// TwinCAT 3 PLC project HalfBROT
// Title: HalfBROT
// Company: BROT
// ProjectVersion: 0.4.4
// ProgramVersion: 3.1.4024.66
// CompilerDefines: VISU_USEPROPERTYINFO
// libraries:
//   AstroBROT, * (BROT)
//   BROTLib, * (BROT)
//   Tc2_MC2, * (Beckhoff Automation GmbH)
//   Tc2_MC2_Drive, * (Beckhoff Automation GmbH)
//   Tc2_Standard, * (Beckhoff Automation GmbH)
//   Tc2_System, * (Beckhoff Automation GmbH)
//   Tc2_Utilities, * (Beckhoff Automation GmbH)
//   Tc3_Module, * (Beckhoff Automation GmbH)
//   VisuDialogs, * (System)
//   VisuSymbols, * (System)
//   VisuSymbols,3.5.10.0,System
// project tree:
//   / GlobalTextList.TcGTLO, VisualizationManager.TcVMO (not stored)
//   POUs/ FB_AxisControl.TcPOU, FB_AzimuthControl.TcPOU, FB_CoverControl.TcPOU, FB_DerotatorControl.TcPOU, FB_ElevationControl.TcPOU, FB_FocusControl.TcPOU, FB_HydraulicsControl.TcPOU, FB_PendantControl.TcPOU, FB_TelescopeAuxiliary.TcPOU
//   VISUs/ Azimuth.TcVIS, Cover.TcVIS, Derotator.TcVIS, Elevation.TcVIS, Focus.TcVIS, Hydraulics.TcVIS
//   GVLs/ Global_Version.TcGVL

// ---- GVLs/Global_Version.TcGVL
{attribute 'qualified_only'}
VAR_GLOBAL CONSTANT
	// Mirrors Beckhoff's own Global_Version.stLibVersion_* pattern (see ST_LibVersion),
	// which only covers Tc2_*/Tc3_* library references, not custom ones -- until now: this
	// GVL uses Beckhoff's own naming exactly, so it merges into a consumer's Global_Version.
	// Kept in sync with <ProjectVersion> in HalfBROT.plcproj at release time.
	stLibVersion_HalfBROT : ST_LibVersion := (
		iMajor := 0,
		iMinor := 4,
		iBuild := 4,
		iRevision := 0,
		nFlags := 1,
		sVersion := '0.4.4'
	);
END_VAR

// ---- POUs/FB_AxisControl.TcPOU
FUNCTION_BLOCK ABSTRACT FB_AxisControl EXTENDS FB_BaseAxis IMPLEMENTS I_Axis
VAR_INPUT
	bMoveAxis				: BOOL;		// Move azimuth to given position
	bTracking				: BOOL;		// enable tracking
	bStopAxis				: BOOL;		// stop the Axis
	fMinPosition			: REAL := 0;
	fMaxPosition			: REAL := 450.0;
	fCalibPosition			: LREAL := 45.0; // // current position of the calibration cam
END_VAR
VAR_OUTPUT
END_VAR
VAR
	fSlewTime				: LREAL;	// time to reach target position

	InDigitalInputs	  AT%I*	: WORD;		// digitale inputs der Endlagen
	InDiagnostic	  AT%I*	: UDINT;	// diagnostic number
	InTorque	 	  AT%I*	: INT;		// derotator torque feedback
	IbSTO		  	  AT%I*	: BOOL;		// STO

	fbAxisCalibration		: MC_SetPosition;

	axisEvent			: FB_EventLog;
	diagnosticEvent		: FB_EventLog;
	
	bDiagnosticError		: BOOL;
	
	fbReadParameter		: MC_ReadParameter;
	bGetLastPosition		: BOOL := TRUE;
	
	calibrationEvent		: FB_Eventlog;
	fTorque			: REAL;	// percentage of the derotator torque
	torqueWarning			: FB_EventLog;	
END_VAR
VAR PERSISTENT
	fLastPosition			: LREAL := -1.0;
END_VAR

PROPERTY isTracking : BOOL
GET
isTracking := fbAxis.isTracking;
END_GET
END_PROPERTY

PROPERTY MoveAxis : BOOL
GET
MoveAxis := bMoveAxis;
END_GET
SET
bMoveAxis := MoveAxis;
END_SET
END_PROPERTY

PROPERTY MoveDone : BOOL
GET
MoveDone := fbAxis.MoveDone;
END_GET
END_PROPERTY

PROPERTY SlewTime : LREAL
GET
SlewTime := fSlewTime;
END_GET
END_PROPERTY

PROPERTY StopAxis : BOOL
GET
StopAxis := bStopAxis;
END_GET
SET
bStopAxis := StopAxis;
END_SET
END_PROPERTY

PROPERTY Tracking : BOOL
GET
Tracking := bTracking;
END_GET
SET
bTracking := Tracking;
END_SET
END_PROPERTY

END_FUNCTION_BLOCK

// ---- POUs/FB_AzimuthControl.TcPOU
FUNCTION_BLOCK FB_AzimuthControl EXTENDS FB_AxisControl
VAR_INPUT
	bBrakeOpen				: BOOL;		// azimuth break is open
END_VAR
VAR_OUTPUT
END_VAR
VAR
	tonReadyDelay		: TON;		// delay until commutator angle is measured
	homeDelay			: FB_TONTP;
	tonTorqueError		: TON := (PT := T#3S);
	tonRestTimer			: TON;
	bAtRest				: BOOL;
END_VAR

(* Azimuth Axis control section
Power must be on and brake must be open for the axis to operate
*)

// generate the ready signal after enabling the drive
tonReadyDelay(IN :=  fbAxis.Enable, PT := T#3000MS, Q=> bReady);

// limit the input position angle
fPosition := LIMIT(fMinPosition, fPosition, fMaxPosition);

// conduct the calibrated signal
bCalibrated := fbAxis.Calibrated;

IF bCalibrated OR bError THEN
	bHomeAxis := FALSE;
	bGetLastPosition := FALSE;
END_IF
	
IF bHomeAxis THEN
	fPosition := fCalibPosition;
END_IF

IF homeDelay.Q THEN
	fPosition := fCalibPosition;
	bMoveAxis := TRUE;
END_IF

// perform a recalibration on the last known position
fbAxisCalibration(
	Axis 		:= axisRef,
	Execute 	:= bGetLastPosition AND fLastPosition>=0.0 AND NOT bCalibrated,
	Position 	:= fLastPosition);

IF fbAxisCalibration.Done THEN
	bGetLastPosition := FALSE;
END_IF

IF bCalibrated THEN
	fLastPosition := fActualPosition;
END_IF

// enable the azimuth if not moved by the power chain. Sorry for the hack
tonRestTimer(IN := bBrakeOpen AND (ABS(axisRef.NcToPlc.ActVelo) < 0.01), PT := T#2S);
// if azimuth at rest or calibrated, allow enabling the azimuth (the brake must still be open, see Enable below)
IF tonRestTimer.Q or bCalibrated THEN
	bAtRest := TRUE;
ELSIF NOT bBrakeOpen THEN
	bAtRest := FALSE;
END_IF
	
// deactivate limit switches on homing
MC_SetAcceptBlockedDriveSignal(
	Axis 	:= axisRef, 
	Enable 	:= bHomeAxis);

fbAxis(	
	Enable 			:= bEnable AND bAtRest AND bBrakeOpen,
	Reset 			:= bReset,
	MoveAxis 		:= bMoveAxis,
	HomeAxis 		:= bHomeAxis,
	StopAxis 		:= bStopAxis,
	Tracking 		:= bTracking,
	Position 		:= fPosition, 
	Velocity 		:= fVelocity,
	Enable_Positive := inDigitalInputs.1 OR bHomeAxis,
	Enable_Negative := inDigitalInputs.0,
	Jog_Forward 	:= bMovePos,
	Jog_Backwards 	:= bMoveNeg,
	bCalibrationCam := NOT inDigitalInputs.1,
	ActualPosition 	=> fActualPosition,
	Error 			=> bError,
	ErrorID 		=> nErrorID,
	AxisRef 		:= axisRef);

IF bSoEReset THEN
	fLastPosition := -1.0;
	fbSoEReset(
		Axis 	:= axisRef,
		Execute := TRUE,
		Timeout := DEFAULT_ADS_TIMEOUT);
 	IF fbSoEReset.Busy THEN
		fbSoEReset(Axis := axisRef, Execute := FALSE);
	ELSE
		bSoEReset := FALSE;
		bReset := TRUE;
	END_IF
END_IF 

IF fbAxis.MoveDone THEN
	bMoveAxis := FALSE;
END_IF

IF fbAxis.HomeDone THEN
	bHomeAxis := FALSE;
END_IF
	
IF fbAxis.ResetDone THEN
	bReset := FALSE;
END_IF

IF fbAxis.StopDone THEN
	bStopAxis := FALSE;
END_IF
bDiagnosticError := FALSE;
IF inDiagnostic < 16#D012 AND inDiagnostic > 16#D014 THEN
	bDiagnosticError :=TRUE;
	nErrorID := inDiagnostic;
END_IF

fbReadParameter(	
	Axis 			:= axisRef, 
	Enable 			:= fbAxis.InMotion, 
	ParameterNumber := MC_AxisParameter.AxisRemainingTimeToGo, 
	ReadMode 		:= E_ReadMode.READMODE_CYCLIC);
IF fbReadParameter.Valid THEN
	fSlewTime := fbReadParameter.Value;
END_IF

fTorque := inTorque / 10.0;
tonTorqueError(IN := ABS(fTorque) > 50.0);

axisEvent(	
	Trigger 		:= bError, 
	Level 			:= ADSLOG_MSGTYPE_ERROR,
	FormatString 	:= 'Azimuth Axis Error: %s',
	OnMessage 		:= NCError_TO_STRING(nErrorID),
	Comm 			:= fbComm);
	
diagnosticEvent(	
	Trigger 		:= bDiagnosticError,
	Level 			:= ADSLOG_MSGTYPE_ERROR,
	FormatString 	:= 'Azimuth Axis Diagnostic Error: %s',
	OnMessage 		:= NCError_TO_STRING(inDiagnostic),
	Comm 			:= fbComm);
	
TorqueWarning(	
	Trigger 		:= tonTorqueError.Q, 
	Level 			:= ADSLOG_MSGTYPE_WARN,
	FormatString 	:= '%s',
	OnMessage 		:= 'Azimuth torque is high.',
	Comm 			:= fbComm);
	
CalibrationEvent(
	Trigger 		:= bCalibrated, 
	Level 			:= ADSLOG_MSGTYPE_HINT,
	FormatString 	:= '%s',
	OnMessage 		:= 'Azimuth axis is calibrated.',
	Comm 			:= fbComm);

PROPERTY InNegLimit : BOOL
GET
InNegLimit := NOT inDigitalInputs.0;
END_GET
END_PROPERTY

PROPERTY InPosLimit : BOOL
GET
InPosLimit := NOT inDigitalInputs.1;
END_GET
END_PROPERTY

END_FUNCTION_BLOCK

// ---- POUs/FB_CoverControl.TcPOU
FUNCTION_BLOCK FB_CoverControl IMPLEMENTS I_MirrorCovers
VAR_INPUT
	// output signals for opening/closing covers	
	OabOpenCover  AT%Q* : ARRAY[1..3] OF BOOL;	// open cover1-3 command
	OabCloseCover AT%Q* : ARRAY[1..3] OF BOOL;   // close cover1-3 command
	
	// telemetry interval
	fTelemetryInterval		: TIME := T#5S;	
END_VAR
VAR_OUTPUT
	bAllOpen			: BOOL;		// all covers are open
	bAllClosed			: BOOL;		// all covers are closed
	bError				: BOOL;		// any cover-driver reports an error
	bWarning			: BOOL;		// warning state of the DC drives
END_VAR
VAR
	fbComm				: I_Comm;
	tonComm 			: TON := (PT:=fTelemetryInterval);	

	bReset				: BOOL;		// resets all drives after an error has occured
	bOpen				: BOOL;		// open the cover in proper order
	bClose				: BOOL;		// close the cover in proper order

	// limit switches
	IabCoverOpen	AT%I* : ARRAY[1..3] OF BOOL;	// limit coper 1 open switch
	IabCoverClosed	AT%I* : ARRAY[1..3] OF BOOL;	// limit coper 1 closed switch
	
	// status
	abCoverOpen			: ARRAY[1..3] OF BOOL;	// cover is open
	abCoverClosed		: ARRAY[1..3] OF BOOL;	// cover is closed
	abCoverError			: ARRAY[1..3] OF BOOL;	// cover has error
	afbCoverEvent			: ARRAY[1..3] OF FB_EventLog;	// cover event
	afbTimeoutEvent : ARRAY[1..3] OF FB_EventLog;	// cover has timeout
	
	tonCover2OpenDelay		: TON := (PT:=T#1S);	// delay timer for opening cover2
	tonCover3CloseDelay 	: TON := (PT:=T#3S);	// dely timer for closing cover3

	srErrorTrigger			: SR;	// trigger for error
	
	fbCoversOpenedEvent		: FB_EventLog; // log if covers are open
	fbCoversClosedEvent		: FB_EventLog; // log if covers are closed
	fbCoversErrorEvent		: FB_EventLog; // Event log for a generic drive error
	fbCoversWarningEvent	: FB_EventLog; // Event log for a generic drive warning
	
	i	: UINT;
END_VAR

(*
This is the control for the two (three) telescope covers. 
The correct order for opening is 1->3->2 and for closing 2->3->1.
GVL Open and close signals are inverted
*)

// close has precedence over open
IF bClose THEN
	bOpen := FALSE;
END_IF

// do stuff for all covers
FOR i := 1 TO 3 BY 1 DO
	// limit switches are inverted
    abCoverOpen[i]   := NOT IabCoverOpen[i];
	abCoverClosed[i] := NOT IabCoverClosed[i];
	
	// errors occur if covers are both opened and closed
	abCoverError[i] := abCoverOpen[i] AND abCoverClosed[i];
END_FOR;

// wait for cover2 until cover3 has left the closed state
tonCover2OpenDelay(IN := bOpen AND NOT abCoverClosed[3]);
// wait for cover3 until cover2 has left the open state
tonCover3CloseDelay(IN := bClose AND NOT abCoverOpen[2]);

// commands
IF bClose THEN
	OabCloseCover[1] := IabCoverClosed[1] AND NOT IabCoverClosed[3];
	OabCloseCover[2] := IabCoverClosed[2];
	OabCloseCover[3] := IabCoverClosed[3] AND tonCover3CloseDelay.Q;
ELSIF bOpen THEN
	OabOpenCover[1] := IabCoverOpen[1];
	OabOpenCover[2] := IabCoverOpen[2] AND tonCover2OpenDelay.Q;
	OabOpenCover[3] := IabCoverOpen[3];			
END_IF

// we are open, if all covers are open
bAllOpen := abCoverOpen[1] AND abCoverOpen[2] AND abCoverOpen[3];
// we are closed, if all covers are closed
bAllClosed := abCoverClosed[1] AND abCoverClosed[2] AND abCoverClosed[3];

// error indicates an axis error on any axis
srErrorTrigger(
	SET1 := abCoverError[1] OR abCoverError[2] OR abCoverError[3],
	RESET := bReset,
	Q1 => bError);

// clear reset, if no error present
IF NOT bError THEN
	bReset := FALSE;
END_IF

IF bAllClosed THEN
	bClose := FALSE;
END_IF

IF bAllOpen THEN
	bOpen := FALSE;
END_IF

fbCoversErrorEvent.OnMessage := 'Cover drive error';
IF bError THEN
	IF abCoverError[3] THEN 
		fbCoversErrorEvent.OnMessage := 'Cover 3 has a drive error.';
	END_IF
	IF abCoverError[2] THEN 
		fbCoversErrorEvent.OnMessage := 'Cover 2 has a drive error.';
	END_IF
	IF abCoverError[1] THEN 
		fbCoversErrorEvent.OnMessage := 'Cover 1 has a drive error.';
	END_IF
END_IF

// send telemetry
tonComm(IN:=TRUE);
IF tonComm.Q THEN // publish new payload every second
	tonComm(IN:=FALSE);
	THIS^._SendTelemetry();	
END_IF

fbCoversErrorEvent(
	Trigger 	:= bError, 
   	Level   	:= ADSLOG_MSGTYPE_ERROR, 
	comm 		:= fbComm);

fbCoversWarningEvent(
	Trigger 	:= bWarning, 
	Level   	:= ADSLOG_MSGTYPE_WARN, 
	comm 		:= fbComm);

// raise an error, if both opened and closed signals are activated
// handle RoboTel differently
afbCoverEvent[1](
	Trigger   	:= abCoverOpen[1] AND abCoverClosed[1],
	Level     	:= ADSLOG_MSGTYPE_ERROR, 
	OnMessage 	:= 'Cover1: limit switch error', 
	comm	 	:= fbComm);

afbCoverEvent[2](
	Trigger   	:= abCoverOpen[2] AND abCoverClosed[2],
    Level     	:= ADSLOG_MSGTYPE_ERROR, 
	OnMessage 	:= 'Cover2: limit switch error', 
	comm      	:= fbComm);

afbCoverEvent[3](
	Trigger   	:= abCoverOpen[3] AND abCoverClosed[3],
	Level     	:= ADSLOG_MSGTYPE_ERROR, 
	OnMessage 	:= 'Cover3: limit switch error', 
	comm 	  	:= fbComm);

//trigger an event, if we encounter a timeout
// handle RoboTel differently
afbTimeoutEvent[1](
	Trigger   	:= FALSE,
	Level     	:= ADSLOG_MSGTYPE_ERROR, 
	OnMessage 	:= 'Cover1: Timeout',
	comm 		:= fbComm);
afbTimeoutEvent[2](
	Trigger   	:= FALSE,
 	Level     	:= ADSLOG_MSGTYPE_ERROR, 
	OnMessage 	:= 'Cover2: Timeout',
	comm 		:= fbComm);
afbTimeoutEvent[3](
	Trigger   	:= FALSE,
	Level     	:= ADSLOG_MSGTYPE_ERROR, 
	OnMessage 	:= 'Cover3: Timeout',
	comm 		:= fbComm);

// Log if we are opened
fbCoversOpenedEvent(
	Trigger   	:= bAllOpen,
	Level     	:= ADSLOG_MSGTYPE_WARN,
	OnMessage 	:= 'All covers are open',
	comm 		:= fbComm);
	
//log if we are closed
fbCoversClosedEvent(
	Trigger   	:= bAllClosed,
	Level     	:= ADSLOG_MSGTYPE_HINT,
	OnMessage 	:= 'All covers are closed',
	comm 		:= fbComm);

METHOD _SendTelemetry : BOOL
VAR_INPUT
END_VAR
IF bAllClosed THEN
	fbComm.Publish('telescope', 'dome', 'AUXILIARY.COVER.REALPOS', '0.0');
ELSIF bAllOpen THEN
	fbComm.Publish('telescope', 'dome', 'AUXILIARY.COVER.REALPOS', '1.0');
ELSE
	fbComm.Publish('telescope', 'dome', 'AUXILIARY.COVER.REALPOS', '0.5');
END_IF
END_METHOD

METHOD Close : BOOL
VAR_INPUT
END_VAR
bOpen := FALSE;
bClose := TRUE;
END_METHOD

PROPERTY Closed : BOOL
GET
Closed := bAllClosed;
END_GET
END_PROPERTY

PROPERTY Error : BOOL
GET
Error := bError;
END_GET
END_PROPERTY

//FB_Init is always available implicitly and it is used primarily for initialization.
//The return value is not evaluated. For a specific influence, you can also declare the
//methods explicitly and provide additional code there with the standard initialization
//code. You can evaluate the return value.
METHOD FB_Init: BOOL
VAR_INPUT
    bInitRetains	: BOOL; // TRUE: the retain variables are initialized (reset warm / reset cold)
    bInCopyCode		: BOOL;  // TRUE: the instance will be copied to the copy code afterward (online change)
	comm			: I_Comm;   
END_VAR
THIS^.fbComm := comm;
END_METHOD

METHOD Open : BOOL
VAR_INPUT
END_VAR
bOpen := TRUE;
bClose := FALSE;
END_METHOD

PROPERTY Opened : BOOL
GET
Opened := bAllOpen;
END_GET
END_PROPERTY

METHOD Reset : BOOL
VAR_INPUT
END_VAR
bReset := TRUE;
Reset := TRUE;
END_METHOD

END_FUNCTION_BLOCK

// ---- POUs/FB_DerotatorControl.TcPOU
FUNCTION_BLOCK FB_DerotatorControl EXTENDS FB_AxisControl
VAR_INPUT
END_VAR
VAR_OUTPUT
END_VAR
VAR
	tonTorqueError		: TON := (PT := T#3S);	// trigger for the torque error
END_VAR

(*
Selection 6
Homing in Endlage:

https://infosys.beckhoff.com/index.php?content=../content/1031/ax5000_usermanual/html/ax5000_homing_hardware_end_position.htm&id=12221
NC-Interface:
PlcToNc-Achsinterface, Bit 8 namens AcceptBlockedDriveSignal im nDeCtrlDWord

SPS-Interface:
TcNc-Lib, siehe SPS-Funktion AxisSetAcceptBlockedDriveSignal in der TwinCAT  PLC Library: NC.
*)

fPosition := LIMIT(fMinPosition, fPosition, fMaxPosition);

IF bEnable AND NOT fbAxis.Calibrated THEN
	bHomeAxis := TRUE;
END_IF

IF fbAxis.Calibrated THEN
	bHomeAxis := FALSE;
	bCalibrated := fbAxis.Calibrated;
END_IF
	
IF bHomeAxis THEN
	fPosition := fCalibPosition;
END_IF

IF fbAxis.ActualPosition > fMaxPosition OR fbAxis.ActualPosition < fMinPosition THEN
	bStopAxis := TRUE;
END_IF

fbAxis(
	enable 			:= bEnable,
	Reset 			:= bReset,
	MoveAxis 		:= bMoveAxis,
	HomeAxis 		:= bHomeAxis,
	StopAxis 		:= bStopAxis,
	HomingMode 		:= MC_ForceCalibration,
	Position 		:= fPosition, 
	Velocity 		:= fVelocity,
	Enable_Positive := fbAxis.ActualPosition < fMaxPosition,
	Enable_Negative := fbAxis.ActualPosition > fMinPosition,
	Jog_Forward 	:= bMovePos,
	Jog_Backwards 	:= bMoveNeg,
	//bCalibrationCam := inDigitalInputs.0,
	isModuloAxis 	:= FALSE,
	Tracking 		:= bTracking,
	ActualPosition 	=> fActualPosition,
	Error 			=> bError,
	ErrorID 		=> nErrorID,
	AxisRef 		:= axisRef);
	
IF fbAxis.MoveDone OR bReset OR bError THEN
	bMoveAxis := FALSE;
END_IF

IF fbAxis.HomeDone OR bReset OR bError THEN
	bHomeAxis := FALSE;
END_IF
	
IF fbAxis.ResetDone THEN
	bReset := FALSE;
END_IF

IF fbAxis.StopDone THEN
	bStopAxis := FALSE;
END_IF

bDiagnosticError := FALSE;
IF inDiagnostic < 16#D012 AND inDiagnostic > 16#D014 THEN
	bDiagnosticError := TRUE;
	nErrorID := inDiagnostic;
	bSoeReset := bReset;
END_IF

bReady := fbAxis.Ready;

fbReadParameter(	
	Axis 			:= axisRef, 
	Enable 			:= fbAxis.InMotion, 
	ParameterNumber := MC_AxisParameter.AxisRemainingTimeToGo, 
	ReadMode 		:= E_ReadMode.READMODE_CYCLIC);
				
IF fbReadParameter.Valid THEN
	fSlewTime := fbReadParameter.Value;
END_IF

IF bSoEReset THEN
	fbSoEReset(
		Axis 	:= axisRef,
		Execute := TRUE,
		Timeout := DEFAULT_ADS_TIMEOUT);
 	IF NOT fbSoEReset.Busy THEN
		fbSoEReset(Axis := axisRef, Execute := FALSE);
		bSoEReset := FALSE;
		bReset := TRUE;
	END_IF
END_IF

fTorque := inTorque / 10.0;
// nominal torque is 3%, max is 25%
tonTorqueError(IN := ABS(fTorque) > 20.0);

axisEvent(	
	Trigger 		:= bError, 
	Level 			:= ADSLOG_MSGTYPE_ERROR,
	FormatString	:= 'Derotator Axis Error: %s',
	OnMessage 		:= NCError_TO_STRING(nErrorID),
	OffMEssage 		:= 'OK',
	OffLevel 		:= ADSLOG_MSGTYPE_HINT,
	Comm			:= fbComm);
	
diagnosticEvent(	
	Trigger 		:= bDiagnosticError, 
	Level 			:= ADSLOG_MSGTYPE_ERROR,
	FormatString	:= 'Derotator Axis Diagnostic Error: %s',
	OnMessage 		:= NCError_TO_STRING(inDiagnostic),
	Comm			:= fbComm);
	
TorqueWarning(	
	Trigger 		:= tonTorqueError.Q, 
	Level 			:= ADSLOG_MSGTYPE_WARN,
	FormatString 	:= '%s',
	OnMessage 		:= 'Derotator torque is high.',
	Comm			:= fbComm);

CalibrationEvent(	
	Trigger 		:= bCalibrated, 
	Level 			:= ADSLOG_MSGTYPE_HINT,
	OnMessage 		:= 'Derotator is calibrated.',
	Comm			:= fbComm);

PROPERTY InNegLimit : BOOL
GET
InNegLimit := inDigitalInputs.1;
END_GET
END_PROPERTY

PROPERTY InPosLimit : BOOL
GET
InPosLimit := inDigitalInputs.0;
END_GET
END_PROPERTY

END_FUNCTION_BLOCK

// ---- POUs/FB_ElevationControl.TcPOU
FUNCTION_BLOCK FB_ElevationControl EXTENDS FB_AxisControl
VAR_INPUT
	fbCovers		: I_MirrorCovers;
	fbBrake			: I_Brake;
END_VAR
VAR_OUTPUT
	bWarning			: BOOL;		// warning condition
END_VAR
VAR
	tonReadyDelay			: TON;	// delay until commutator angle is measured
	enableTrigger			: F_TRIG;	// disable trigger for hydraulics
	brakeEvent				: FB_Eventlog;
	highElevationEvent		: FB_Eventlog;
	lowElevationEvent		: FB_Eventlog;
	tonTorqueTimer				: TON;		// timer to trigger a warning if torque is high
END_VAR

// limit the position input to a sane value
fPosition := LIMIT(0.0, fPosition, 90.0);

//if we enable the axis, we have to open the brake first
IF bEnable THEN
	IF NOT bCalibrated THEN
		fbCovers.Open();
		IF fbCovers.Opened THEN
			fbBrake.OpenBrake();
		END_IF
	ELSE
		fbBrake.OpenBrake();
	END_IF
	
END_IF

enableTrigger(CLK := bEnable);
// close the brake on the falling edge of the enable signal
IF enableTrigger.Q THEN
	fbBrake.CloseBrake();
END_IF

IF fbAxis.Calibrated OR bError THEN
	bHomeAxis := FALSE;
END_IF

bCalibrated := fbAxis.Calibrated;

IF bHomeAxis THEN
	fPosition := fCalibPosition;
	bMoveAxis := FALSE;
	bTracking := FALSE;
END_IF

IF bMoveAxis THEN
	bTracking := FALSE;
END_IF

// if NOT Enabled and ActVelo>1 then issue a warning
bWarning := NOT bEnable AND axisRef.NcToPlc.ActVelo>2.0;

// deactivate limit switches on homing
MC_SetAcceptBlockedDriveSignal(
	Axis := axisRef, 
	Enable := bHomeAxis);
	
fbAxis(
	Enable 			:= bEnable AND fbBrake.BrakeOpen,
	Reset 			:= bReset,
	MoveAxis 		:= bMoveAxis,
	HomeAxis 		:= bHomeAxis,
	StopAxis 		:= bStopAxis,
	Tracking 		:= bTracking,
	Position 		:= fPosition, 
	Velocity 		:= fVelocity,
	Enable_Positive := inDigitalInputs.0 OR bHomeAxis,
	Enable_Negative := inDigitalInputs.1,
	Jog_Forward 	:= bMovePos,
	Jog_Backwards 	:= bMoveNeg,
	bCalibrationCam := NOT inDigitalInputs.0,
	ActualPosition 	=> fActualPosition,
	Error 			=> bError,
	ErrorID 		=> nErrorID,
	AxisRef 		:= axisRef);

IF fbAxis.MoveDone THEN
	bMoveAxis := FALSE;
END_IF

IF fbAxis.HomeDone THEN
	bHomeAxis := FALSE;
END_IF
	
IF fbAxis.ResetDone THEN
	bReset := FALSE;
END_IF

IF fbAxis.StopDone THEN
	bStopAxis := FALSE;
END_IF

bDiagnosticError := FALSE;
IF inDiagnostic < 16#D012 AND inDiagnostic > 16#D014 THEN
	bDiagnosticError :=TRUE;
	nErrorID := inDiagnostic;
END_IF

fbAxisCalibration(
	Axis 		:= axisRef,
	Execute 	:= bGetLastPosition AND fLastPosition>=0.0 AND NOT bCalibrated,
	Position 	:= fLastPosition);

IF fbAxisCalibration.Done THEN
	bGetLastPosition := FALSE;
END_IF

IF bCalibrated THEN
	fLastPosition := fActualPosition;
END_IF

IF bSoEReset THEN
	fLastPosition := -1.0;
	fbSoEReset(
		Axis := axisRef,
		Execute := TRUE,
		Timeout := DEFAULT_ADS_TIMEOUT);
 	IF NOT fbSoEReset.Busy THEN
		fbSoEReset(Axis := axisRef, Execute := FALSE);
		bSoEReset := FALSE;
		bReset := TRUE;
	END_IF
END_IF 

tonReadyDelay(IN :=  fbBrake.BrakeOpen, PT := T#6000MS, Q=> bReady);

fbReadParameter(	
	Axis 			:= axisRef, 
	Enable 			:= fbAxis.InMotion, 
	ParameterNumber := MC_AxisParameter.AxisRemainingTimeToGo, 
	ReadMode 		:= E_ReadMode.READMODE_CYCLIC);
				
IF fbReadParameter.Valid THEN
	fSlewTime := fbReadParameter.Value;
END_IF

fTorque := inTorque / 10.0;
tonTorqueTimer(IN := ABS(fTorque) > 50.0, PT := T#1000MS);
		
axisEvent(	
	Trigger 		:= bError, 
	Level 			:= ADSLOG_MSGTYPE_ERROR,
	FormatString 	:= 'Elevation Axis Error: %s',
	OnMessage 		:= NCError_TO_STRING(nErrorID), 
	comm 			:= fbComm);

diagnosticEvent(	
	Trigger 		:= bDiagnosticError,
	Level 			:= ADSLOG_MSGTYPE_ERROR,
	FormatString 	:= 'Elevation Axis Diagnostic Error: %s',
	OnMessage 		:= NCError_TO_STRING(inDiagnostic), 
	comm 			:= fbComm);

highElevationEvent(	
	Trigger 		:= bCalibrated AND fActualPosition > 85.0, 
	Level 			:= ADSLOG_MSGTYPE_WARN,
	FormatString 	:= 'High Elevation: %s',
	OnMessage 		:= LREAL_TO_FMTSTR(fActualPosition, 2, TRUE), 
	comm 			:= fbComm);

lowElevationEvent(	
	Trigger 		:= bCalibrated AND fActualPosition < 5.0, 
	Level 			:= ADSLOG_MSGTYPE_WARN,
	FormatString 	:= 'Low Elevation: %s',
	OnMessage 		:= LREAL_TO_FMTSTR(fActualPosition, 2, TRUE), 
	comm 			:= fbComm);
				
brakeEvent( 
	Trigger 		:= NOT bEnable AND fbBrake.BrakeOpen, 
	Level 			:= ADSLOG_MSGTYPE_WARN,
	FormatString 	:= '%s',
	OnMessage 		:= 'Brake was opened without elevation axis enabled!', 
	comm 			:= fbComm); 

torqueWarning(	
	Trigger 		:= tonTorqueTimer.Q, 
	Level 			:= ADSLOG_MSGTYPE_WARN,
	FormatString 	:= '%s',
	OnMessage 		:= 'Elevation torque is high.', 
	comm 			:= fbComm);
	
calibrationEvent(
	Trigger 		:= bCalibrated,
	Level 			:= ADSLOG_MSGTYPE_HINT,
	OnMessage 		:= 'Elevation is calibrated.', 
	comm 			:= fbComm);

PROPERTY InNegLimit : BOOL
GET
InNegLimit := NOT inDigitalInputs.1;
END_GET
END_PROPERTY

PROPERTY InPosLimit : BOOL
GET
InPosLimit := NOT inDigitalInputs.0;
END_GET
END_PROPERTY

END_FUNCTION_BLOCK

// ---- POUs/FB_FocusControl.TcPOU
FUNCTION_BLOCK FB_FocusControl EXTENDS FB_BaseAxis IMPLEMENTS I_Focus
VAR_INPUT
	fMinPosition		: LREAL := 0;	// minimum position
	fMaxPosition		: LREAL := 100;	// maximum position
	eTelescopeMode		: E_TelescopeMode;
	fHomingPosition		: LREAL := 92.02; // 104.02 - 12.00 	// reference position for homing
	fTolerance			: LREAL := 0.005;
	
	// telemetry interval
	fTelemetryInterval		: TIME := T#5S;
	ptFocusDelay			: TIME := T#500MS;
	ptBrakeDelay			: TIME := T#4S;	
END_VAR
VAR_OUTPUT
	bFocusUnlocked		: BOOL;
END_VAR
VAR
	bMoveAxis			: BOOL;		// move the axis to new position
	ObFocusUnlock AT%Q* : BOOL;		// whether focus is unlocked
	tonFocusDelay		: TON;
	tonBrakeDelay		: TON;
	bManualUnlock		: BOOL;		// manual override to unlock the focus
	tonComm 			: TON := (PT:=fTelemetryInterval);
	//getlastposition:	BOOL := TRUE;
	fbAxisEvent			: FB_EventLog;
	fbCalibrationEvent	: FB_EventLog;
	eHomingMode			: MC_HOMINGMODE := MC_DefaultHoming;
	fbSetPosition		: MC_SetPosition;
	
	IbLimitNear    AT%I*: BOOL;	// DIN29 3.4
	IbLimitFar     AT%I*: BOOL;	// DIN30 3.5
	refAxis			: AXIS_REF;
END_VAR
VAR PERSISTENT
	fLastPposition		: LREAL := -1.0;
END_VAR

(*
Focus Control Unit
spindle gear: 5mm
brake: 86 61103H00 Var. 0005 Index C; 24VDC geglattet 0,25 A P1672/R7
motor: Faulhaber ; Schönaich ; 3557K024CR; 454  431 ; Made in germany ==> 5300 rpm
gear: Faulhaber ; MINIMOTOR SA ; swiss made ; 38/1S  43:1 ; 033896  503
Focus is locked by default
70,8W; 0,100A no load current; 2,0 Terminal resistance; 1,950A max Current 
*)

// limit to sane positions
fPosition := LIMIT(fMinPosition, fPosition, fMaxPosition);

// focus is unlocked if enabled or manually unlocked and no eror
ObFocusUnlock := (bManualUnlock OR bEnable) AND NOT bError;

// wait until the focus is unlocked for n milliseconds
tonFocusDelay(IN := ObFocusUnlock, PT := ptFocusDelay, Q => bFocusUnlocked);
// wait for brake until we are at rest
tonBrakeDelay(IN := NOT fbAxis.Busy AND fbAxis.StandStill, PT := ptBrakeDelay);

// if we are on automatic mode then position the focus
IF eTelescopeMode = E_TelescopeMode.automatic AND NOT bManualUnlock THEN
	IF fbAxis.calibrated THEN
		IF ABS(fPosition - fActualPosition) > fTolerance THEN
			IF fbAxis.Ready THEN
				bMoveAxis := TRUE;
			ELSE
				bEnable := TRUE;
			END_IF
		END_IF
		// disable the drive and lock the brake, if we stand for more than n seconds
		IF tonBrakeDelay.Q THEN
			bEnable := FALSE;
		END_IF
		// store actual position, if we are calibrated and locked
		IF NOT ObFocusUnlock THEN
			fLastPposition := fActualPosition;
		END_IF
	ELSE // not calibrated
		IF fbAxis.Ready THEN
			bHomeAxis := TRUE;
		END_IF
	END_IF
END_IF

IF bHomeAxis THEN
	IF fLastPposition > 0.0 THEN
		eHomingMode := MC_ForceCalibration; // MC_Direct
		fPosition := fLastPposition;
		fbSetPosition.Execute := TRUE;
	ELSE
		eHomingMode := MC_DefaultHoming;
		fPosition := fHomingPosition;
		fbSetPosition.Execute := FALSE;
	END_IF
ELSE
	fbSetPosition.Execute := FALSE;	
END_IF

// deactivate limit switches on homing
MC_SetAcceptBlockedDriveSignal(Axis := refAxis, enable := bHomeAxis);
fbSetPosition(Axis := refAxis, Position := fLastPposition);
		
fbAxis(	
	enable 			:= bFocusUnlocked,
	Reset 			:= bReset,
	moveAxis 		:= bMoveAxis AND bFocusUnlocked,
	homeAxis 		:= bHomeAxis AND bFocusUnlocked,
	homingMode 		:= eHomingMode,
	Position 		:= fPosition,
	Velocity 		:= fVelocity,
	enable_Positive := NOT IbLimitFar OR bHomeAxis,
	enable_Negative := NOT IbLimitNear,
	Jog_Forward 	:= bMovePos AND bFocusUnlocked,
	Jog_Backwards 	:= bMoveNeg AND bFocusUnlocked,
	bCalibrationCam := IbLimitFar,
	ActualPosition 	=> fActualPosition,
	Error 			=> bError,
	ErrorID 		=> nErrorID,
	axisRef 		:= refAxis);	

IF fbAxis.MoveDone THEN
	bMoveAxis := FALSE;
END_IF

IF fbAxis.HomeDone THEN
	bHomeAxis := FALSE;
	bEnable := FALSE;
	fLastPposition := fPosition;
END_IF
	
IF fbAxis.ResetDone THEN
	bReset := FALSE;
END_IF

IF fbAxis.calibrated OR bError THEN
	bHomeAxis := FALSE;
END_IF

IF bError THEN
	fLastPposition := -1.0;
	//focusAxis.calibrated := FALSE;
	bCalibrated := FALSE;
END_IF

bCalibrated := fbAxis.calibrated;
bReady := fbAxis.Ready AND fbAxis.StandStill OR NOT ObFocusUnlock;

// send telemetry
tonComm(IN:=TRUE);
IF tonComm.Q THEN // publish new payload every 5 seconds
	tonComm(IN:=FALSE);
	THIS^.SendTelemetry();	
END_IF

HandleEvents();

METHOD PROTECTED HandleEvents : BOOL
VAR_INPUT
END_VAR
fbAxisEvent(	
	Trigger 		:= fbAxis.Error, 
	Level 			:= ADSLOG_MSGTYPE_ERROR,
	FormatString	:= 'Focus Axis Error: %S',
	OnMessage 		:= NCError_TO_STRING(nErrorID),
	OffMEssage 		:= 'OK',
	OffLevel 		:= ADSLOG_MSGTYPE_HINT,
	comm 			:= fbComm);

fbCalibrationEvent(
	Trigger 		:=	bCalibrated,
	Level 			:=	ADSLOG_MSGTYPE_HINT,
	OnMessage 		:= 'Focus is calibrated.',
	comm 			:= fbComm);
END_METHOD

PROPERTY PUBLIC InNegLimit : BOOL
GET
InNegLimit := IbLimitNear;
END_GET
END_PROPERTY

PROPERTY PUBLIC InPosLimit : BOOL
GET
InPosLimit := IbLimitFar;
END_GET
END_PROPERTY

METHOD PROTECTED SendTelemetry : BOOL
VAR_INPUT
END_VAR
// > FOCUS
// POWER_STATE
// for now we always return that it's powered on
//IF THIS^.Enable THEN
fbComm.Publish('telescope', 'dome', 'POSITION.INSTRUMENTAL.FOCUS.POWER_STATE', '1.0');
//ELSE
//	fbComm.Publish('telescope', 'dome', 'POSITION.INSTRUMENTAL.FOCUS.POWER_STATE', '0.0');
//END_IF
//REFERENCED
IF THIS^.Calibrated THEN
	fbComm.Publish('telescope', 'dome', 'POSITION.INSTRUMENTAL.FOCUS.REFERENCED', '1.0');
ELSE
	fbComm.Publish('telescope', 'dome', 'POSITION.INSTRUMENTAL.FOCUS.REFERENCED', '0.0');
END_IF
//ERROR_STATE
IF THIS^.Error THEN
	fbComm.Publish('telescope', 'dome', 'POSITION.INSTRUMENTAL.FOCUS.ERROR_STATE', UDINT_TO_STRING(THIS^.ErrorID));
ELSE
	fbComm.Publish('telescope', 'dome', 'POSITION.INSTRUMENTAL.FOCUS.ERROR_STATE', '0');
END_IF
//MOTION_STATE
IF THIS^.Busy THEN
	fbComm.Publish('telescope', 'dome', 'POSITION.INSTRUMENTAL.FOCUS.MOTION_STATE', '1');
ELSE
	fbComm.Publish('telescope', 'dome', 'POSITION.INSTRUMENTAL.FOCUS.MOTION_STATE', '0');
END_IF
fbComm.Publish('telescope', 'dome', 'POSITION.INSTRUMENTAL.FOCUS.CURRPOS', LREAL_TO_STRING(THIS^.ActualPosition));
fbComm.Publish('telescope', 'dome', 'POSITION.INSTRUMENTAL.FOCUS.REALPOS', LREAL_TO_STRING(THIS^.ActualPosition));
fbComm.Publish('telescope', 'dome', 'POSITION.INSTRUMENTAL.FOCUS.TARGETPOS', LREAL_TO_STRING(THIS^.Position));
fbComm.Publish('telescope', 'dome', 'POSITION.INSTRUMENTAL.FOCUS.TARGETDISTANCE', LREAL_TO_STRING(ABS(THIS^.ActualPosition-THIS^.Position)));
fbComm.Publish('telescope', 'dome', 'POSITION.INSTRUMENTAL.FOCUS.CURRSPEED', LREAL_TO_STRING(THIS^.Velocity));
END_METHOD

END_FUNCTION_BLOCK

// ---- POUs/FB_HydraulicsControl.TcPOU
FUNCTION_BLOCK FB_HydraulicsControl IMPLEMENTS I_Hydraulics, I_Brake
VAR_INPUT
	bEnable				: BOOL := FALSE;	// start the hydraulics
	bReset				: BOOL;				// reset any hydraulics error
	bManualSuction		: BOOL;				// manual override to start the suction pump
	bManualPumpStop		: BOOL;				// manual override to stop the pump
	bBrakeClearing		: BOOL;				// external clearing for brakes
	bAzimutLimitSwitch	: BOOL;				// external signal for azimuth limit switch
	nMinPanLevel		: INT := 0;			// minimum oil level from sensor
	nMaxPanLevel		: INT := 16383;		// maximum oil level from sensor
	fMinPanPercent		: REAL := 0;		// oil level percentage to be seen as empty
	fMaxPanPercent		: REAL := 90;		// oil level percentage to be seen as full
	bOpenBrake			: BOOL := FALSE;	// command to open the brake
	bCloseBrake			: BOOL;				// command to open the brake
END_VAR
VAR_OUTPUT
	bBrakeOpen			: BOOL;				// status of the brake: is the brake open?
	bBrakeClosed		: BOOL;				// is the brake closed?
	bPressureFailure	: BOOL;				// pump is running, but the pressure remains low
	bSuctionFailure		: BOOL;				// suction was started, but it is not running
	bHydraulicsFailure	: BOOL;				// main pump is running but suction has a timeout
	bMainPumpFailure	: BOOL;
	bOilLow				: BOOL;				// oil is low
	bOilHigh			: BOOL;				// oil is high (unused?)
	bOilPressureOK		: BOOL;				// oil pressure is 25 bars
	bOilWarning			: BOOL;				// oil is on reserve
	bOilFilterDirty		: BOOL;				// oil filter is dirty
	bOilCold			: BOOL;				// oil is below 10°C
	bOilHot				: BOOL;				// oil is above 50°C
	bOilPanMaximum		: BOOL;				// swimmer
	bPumpRunning		: BOOL;				// main pump is running
	bSuctionRunning 	: BOOL := FALSE;	// suction pump is running
	bError				: BOOL;				// error condition
END_VAR
VAR
	fbComm				: I_Comm;
 
	IbOilLow			AT%I* : BOOL;	// 2.1
	IbOilHigh			AT%I* : BOOL;	// ?
	IbOilPressureOK		AT%I* : BOOL;	// 2.3
	IbOilHot			AT%I* : BOOL;	// 2.4
	IbOilCold			AT%I* : BOOL;	// 2.5
	IbOilFilterDirty	AT%I* : BOOL;	// 2.6
	IbPumpRunning		AT%I* : BOOL;	// 2.7
	IbSuctionRunning	AT%I* : BOOL;	// 2.8
	InOilLevel			AT%I* : INT;	//BT2
	IbOilpanMaximum		AT%I* : BOOL;	//DIN39 4.6
	IbOilReserve		AT%I* : BOOL;	//DIN40 4.7
	ObOilPumpEnable		AT%Q* : BOOL;	//DOUT4 0.3
	ObOilSuctionEnable	AT%Q* : BOOL; //DOUT5 0.4	
	ObBrakeAzEl			AT%Q* : BOOL;	// brake set
	ObResetOilPump		AT%Q* : BOOL;
	ObResetSuctionPump	AT%Q* : BOOL;
	
	tonPressureWatchdog	: TON;				// monitors the pressure of the pump is running
	tonSuctionWatchdog	: TON;				// monitors the activation of the suction pump
	tonMainPumpWatchdog	: TON;				// monitors the activation of the main pump			
	tonHydraulicsWatchdog	: TON;				// watch the hydraulics and suction pumps
	
	rsOilPumpState		: RS;				// represents the state of the main pump
	
	rsBrakeState		: RS;				// represents the state of the brake
	tonBrakeOpenDelay	: TON;				// wait for the brake to open after pressure has been established
	tonBrakeOpenedDelay	: TON;				// report brake opend after a short delay
	tonPressureLossDelay	: TON;				// debounce for loss of oil pressure, which closes the brake

	srErrorState			: SR;				// error state (set dominant)
	srSuctionTrigger		: SR;				// trigger for suction pump
	tonHydraulicsOffTimer	: TON  := (PT := T#300S);	// timer to shut off hydraulics after break was closed
	fbOffTrigger			: F_TRIG;
	fOilLevel			: REAL;
	fLastOilLevel		: REAL;
	hydraulicsLog,
	pumpLog,
	reserveLog,
	oilLowLog,
	filterLog,
	oilMaxLog,
	overTemperatureLog,
	underTemperatureLog,
	suctionLog,
	hydraulicsFailureLog,
	brakeClearingWarning,
	brakeHydraulicsWarning,
	brakeWarning: FB_EventLog;
	
	// measures the operating cycle of the suction pump
	statusWord, lastStatus:	UDINT;
END_VAR

(* 
Main control Logic for the Hydraulics system
* power on delay for main pump and suction pump
* start main pump if main control is ready (button pressed or remote)
* start suction pump if maximum in pan is reached
* suction pump runs until the oil level is below fMinPanPercent
* stop main pump if oil is low
* stop main pump if pressure fails for 30 seconds
*)

// get values from sensors
bOilLow 		:= NOT IbOilLow;
bOilHigh 		:= NOT IbOilHigh;
bOilWarning 	:= IbOilReserve;
bOilPressureOK 	:= IbOilPressureOK;
bOilFilterDirty := NOT IbOilFilterDirty;
bOilCold 		:= NOT IbOilCold;
bOilHot 		:= IbOilHot;
//oil_level 			:= F_YREAL(in_oil_level, 0, 16383, 0.0, 5.0);
fOilLevel		:= F_YREAL(inOilLevel, nMinPanLevel, nMaxPanLevel, 0, 100, cut := FALSE); 
bOilPanMaximum	:= IbOilpanMaximum;
bPumpRunning 	:= IbPumpRunning;
bSuctionRunning := IbSuctionRunning;

// reset pumps
ObResetOilPump     := bReset;
ObResetSuctionPump := bReset;

// error state?
srErrorState(
	SET1  := bPressureFailure OR bSuctionFailure OR bHydraulicsFailure OR bOilLow OR bMainPumpFailure,
	RESET := bReset,
	Q1    => bError);
			
// clear reset, if no error present
IF NOT bError THEN
	bReset := FALSE;
END_IF

// pump state
rsOilPumpState(
	SET    := bEnable,
	RESET1 := NOT bEnable OR bError OR bManualPumpStop OR IbOilpanMaximum);

// switch oil pump
ObOilPumpEnable := rsOilPumpState.Q1;

(* This section controls the hydraulic brake responsible for azimuth and elevation.
The brake needs oil pressure to stay open. There is no brake feedback input, so the
brake state is inferred from the output, the pump and the oil pressure.
The elevation is balanced, but the brake should only be opened, if the elevation drive is activated concurrently.
*)

// losing the oil pressure with the pump running closes the brake
tonPressureLossDelay(
	IN := bPumpRunning AND NOT bOilPressureOK,
	PT := T#2S);

// close the brake if the pump is not running or the pressure is lost
IF bCloseBrake OR NOT bPumpRunning OR tonPressureLossDelay.Q THEN
	bOpenBrake := FALSE;
END_IF

// wait for pressure to build up (hack for oil_pressure_ok)
tonBrakeOpenDelay(
	IN := bPumpRunning AND bOilPressureOK,
	PT := T#3S);
		
rsBrakeState(
	SET    := tonBrakeOpenDelay.Q AND bOpenBrake AND bBrakeClearing,
	RESET1 := bAzimutLimitSwitch OR bCloseBrake OR NOT bPumpRunning OR tonPressureLossDelay.Q OR NOT bBrakeClearing,
	Q1     => ObBrakeAzEl);

// signal that the brake is open after one second
tonBrakeOpenedDelay(
	IN := rsBrakeState.Q1, 
	PT := T#1000MS,
	Q  => bBrakeOpen);

// brake closed?
bBrakeClosed := NOT bBrakeOpen;
IF bBrakeClosed THEN
	bCloseBrake := FALSE;
END_IF

// turn off the hydraulics if the brake is closed and the pump is still running
tonHydraulicsOffTimer(IN := bBrakeClosed AND bEnable );
fbOffTrigger(CLK := tonHydraulicsOffTimer.Q);
IF tonHydraulicsOffTimer.Q THEN
	bEnable := FALSE;
END_IF

(* This is the end of the brake control section *)

srSuctionTrigger(
	SET1  := bOilPanMaximum OR fOilLevel>fMaxPanPercent,
	RESET := fOilLevel<fMinPanPercent);
ObOilSuctionEnable := srSuctionTrigger.Q1 OR bManualSuction;					
tonSuctionWatchdog(
	IN := ObOilSuctionEnable AND NOT bSuctionRunning,
	PT := T#15S,
	Q  => bSuctionFailure);
					
tonPressureWatchdog(
	IN := ObOilPumpEnable AND	NOT bOilPressureOK,
	PT := T#30S,
	Q  => bPressureFailure);
// inherited unchanged from the STELLA1 control, purpose not documented (see #10): error if the main pump
// runs for 140 s without the suction pump running
tonHydraulicsWatchdog(
	IN := bPumpRunning AND NOT bSuctionRunning,
	PT := T#140S,
	Q  => bHydraulicsFailure);

tonMainPumpWatchdog(
	IN := ObOilPumpEnable AND NOT bPumpRunning,
	PT := T#10S,
	Q  => bMainPumpFailure);

statusWord.0 := bOilLow;
statusWord.1 := bOilHigh;
statusWord.2 := bOilWarning;
statusWord.3 := bOilPressureOK;
statusWord.4 := bOilFilterDirty;
statusWord.5 := bOilCold;
statusWord.6 := bOilHot;
statusWord.7 := bBrakeOpen;
statusWord.8 := bBrakeClearing;
statusWord.9 := bPumpRunning;
statusWord.10 := bSuctionRunning;
statusWord.11 := bOilPanMaximum;
statusWord.12 := ObOilPumpEnable;
statusWord.13 := ObOilSuctionEnable;
IF ABS(fLastOilLevel - fOilLevel) > 5 THEN
	statusWord.15 := TRUE;
	fLastOilLevel := fOilLevel;
ELSE
	statusWord.15 := FALSE;
END_IF

IF statusWord<>LastStatus THEN // publish new payload every second
	LastStatus := statusWord;
	fbComm.Publish('hydraulics', 'base', 'OilLow',		BOOL_TO_STRING(bOilLow));
	fbComm.Publish('hydraulics', 'base', 'OilHigh',		BOOL_TO_STRING(bOilHigh));
	fbComm.Publish('hydraulics', 'base', 'OilMaximum',	BOOL_TO_STRING(bOilPanMaximum));
	fbComm.Publish('hydraulics', 'base', 'OilReserve',	BOOL_TO_STRING(bOilWarning));
	fbComm.Publish('hydraulics', 'base', 'OilPressureOK', BOOL_TO_STRING(bOilPressureOK));
	fbComm.Publish('hydraulics', 'base', 'OilFilterDirty',BOOL_TO_STRING(bOilFilterDirty));
	fbComm.Publish('hydraulics', 'base', 'OilCold',		BOOL_TO_STRING(bOilCold));
	fbComm.Publish('hydraulics', 'base', 'OilHot',		BOOL_TO_STRING(bOilHot));
	fbComm.Publish('hydraulics', 'base', 'BrakeOpen',		BOOL_TO_STRING(bBrakeOpen));
	fbComm.Publish('hydraulics', 'base', 'BrakeClearing',	BOOL_TO_STRING(bBrakeClearing));
	fbComm.Publish('hydraulics', 'base', 'PumpRunning',	BOOL_TO_STRING(bPumpRunning));
	fbComm.Publish('hydraulics', 'base', 'SuctionRunning',BOOL_TO_STRING(bSuctionRunning));
	fbComm.Publish('hydraulics', 'base', 'OilLevel',		REAL_TO_STRING(fOilLevel));
	fbComm.Publish('hydraulics', 'base', 'StatusWord',	UDINT_TO_STRING(statusWord));
END_IF

			  
hydraulicsLog(
	Trigger 		:= bPressureFailure OR bMainPumpFailure,
	Level 			:= ADSLOG_MSGTYPE_ERROR,
	FormatString 	:= 'Main hydraulics pump / pressure: %s',
	OnMessage 		:= 'FAILURE',
	OffMessage 		:= 'OK',
	OffLevel 		:= ADSLOG_MSGTYPE_HINT, 
	comm 			:= fbComm);

pumpLog(
	Trigger 		:= bPumpRunning,
	Level 			:= ADSLOG_MSGTYPE_HINT,
	FormatString 	:= 'Main hydraulics pump: %s',
	OnMessage 		:= 'START',
	OffMessage 		:= 'STOP',
	OffLevel 		:= ADSLOG_MSGTYPE_HINT, 
	comm 			:= fbComm);
	
reserveLog(
	Trigger 		:= bOilWarning,
	Level 			:= ADSLOG_MSGTYPE_WARN,
	FormatString 	:= 'oil reserve: %s',
	OnMessage 		:= 'LOW',
	OffMessage 		:= 'OK',
	OffLevel 		:= ADSLOG_MSGTYPE_HINT, 
	comm	 		:= fbComm);

oilLowLog(
	Trigger 		:= bOilLow,
	Level 			:= ADSLOG_MSGTYPE_ERROR,
	FormatString 	:= 'oil level: %s',
	OnMessage 		:= 'LOW',
	OffMessage 		:= 'OK',
	OffLevel 		:= ADSLOG_MSGTYPE_HINT, 
	comm 			:= fbComm);

oilMaxLog(
	Trigger 		:= bOilPanMaximum,
	Level 			:= ADSLOG_MSGTYPE_ERROR,
	FormatString 	:= 'oil level: %s',
	OnMessage 		:= 'MAXIMUM',
	OffMessage 		:= 'OK',
	OffLevel 		:= ADSLOG_MSGTYPE_HINT, 
	comm 			:= fbComm);	
				
filterLog(
	Trigger 		:= bOilFilterDirty,
	Level 			:= ADSLOG_MSGTYPE_WARN,
	FormatString 	:= 'Hydraulics Filter is %s',
	OnMessage 		:= 'dirty.', 
	comm 			:= fbComm);

overTemperatureLog(
	Trigger 		:= bOilHot,
	Level 			:= ADSLOG_MSGTYPE_WARN,
	FormatString 	:= 'Hydraulics Temperature is %s',
	OnMessage 		:= 'high.', 
	comm 			:= fbComm);
				
underTemperatureLog(
	Trigger 		:= bOilCold,
	Level 			:= ADSLOG_MSGTYPE_WARN,
	FormatString 	:= 'Hydraulics Temperature is %s',
	OnMessage 		:= 'low.', 
	comm 			:= fbComm);

suctionLog(
	Trigger 		:= bSuctionFailure,
	Level 			:= ADSLOG_MSGTYPE_ERROR,
	FormatString 	:= 'suction pump: %s',
	OnMessage 		:= 'FAILURE',
	OffMessage 		:= 'OK',
	OffLevel 		:= ADSLOG_MSGTYPE_HINT, 
	comm 			:= fbComm);

hydraulicsFailureLog(
	Trigger 		:= bHydraulicsFailure,
	Level 			:= ADSLOG_MSGTYPE_ERROR,
	FormatString 	:= 'suction pump while running main pump: %s',
	OnMessage 		:= 'FAILURE',
	OffMessage 		:= 'OK',
	OffLevel 		:= ADSLOG_MSGTYPE_HINT, 
	comm 			:= fbComm);
				
brakeClearingWarning(
	Trigger 		:= NOT bBrakeClearing AND bOpenBrake,
	Level 			:= ADSLOG_MSGTYPE_WARN,
	FormatString 	:= '%s',
	OnMessage 		:= 'Cannot open brake without brake clearing.', 
	comm 			:= fbComm);

brakeWarning(	
	Trigger 		:= bBrakeOpen,
	Level 			:= ADSLOG_MSGTYPE_WARN,
	FormatString 	:= '%s',
	OnMessage 		:= 'Brake is open.',
	OffMessage 		:= 'Brake is closed.', 
	comm 			:= fbComm);

brakeHydraulicsWarning(
	Trigger 		:= NOT bEnable AND bOpenBrake,
	Level 			:= ADSLOG_MSGTYPE_WARN,
	FormatString 	:= '%s',
	OnMessage 		:= 'Cannot open brake without running hydraulics.', 
	comm 			:= fbComm);

PROPERTY BrakeOpen : BOOL
GET
BrakeOpen := bBrakeOpen;
END_GET
END_PROPERTY

METHOD CloseBrake : BOOL
VAR_INPUT
END_VAR
// close the brake
bCloseBrake := TRUE;

RETURN(bBrakeClosed);
END_METHOD

PROPERTY Enable : BOOL
GET
Enable := bEnable;
END_GET
SET
bEnable := Enable;
END_SET
END_PROPERTY

PROPERTY Error : BOOL
GET
Error := bError;
END_GET
END_PROPERTY

//FB_Init is always available implicitly and it is used primarily for initialization.
//The return value is not evaluated. For a specific influence, you can also declare the
//methods explicitly and provide additional code there with the standard initialization
//code. You can evaluate the return value.
METHOD FB_Init: BOOL
VAR_INPUT
    bInitRetains	: BOOL; // TRUE: the retain variables are initialized (reset warm / reset cold)
    bInCopyCode		: BOOL;  // TRUE: the instance will be copied to the copy code afterward (online change)
	comm			: I_Comm;
END_VAR
THIS^.fbComm := comm;
END_METHOD

PROPERTY ManualStartSuction : BOOL
GET
ManualStartSuction := bManualSuction;
END_GET
SET
bManualSuction := ManualStartSuction;
END_SET
END_PROPERTY

PROPERTY ManualStopPump : BOOL
GET
ManualStopPump := bManualPumpStop;
END_GET
SET
bManualPumpStop := ManualStopPump;
END_SET
END_PROPERTY

PROPERTY OilPressureOK : BOOL
GET
OilPressureOK := bOilPressureOK;
END_GET
END_PROPERTY

METHOD OpenBrake : BOOL
VAR_INPUT
END_VAR
// start the pump
bEnable := TRUE;
// open the brake
IF bOilPressureOK THEN
	bOpenBrake := TRUE;
END_IF;
RETURN(bBrakeOpen);
END_METHOD

PROPERTY PumpRunning : BOOL
GET
PumpRunning := bPumpRunning;
END_GET
END_PROPERTY

METHOD Reset : BOOL
bReset := TRUE;
END_METHOD

PROPERTY SuctionRunning : BOOL
GET
SuctionRunning := bSuctionRunning;
END_GET
END_PROPERTY

END_FUNCTION_BLOCK

// ---- POUs/FB_PendantControl.TcPOU
FUNCTION_BLOCK FB_PendantControl
VAR_INPUT
	fbCovers			: REFERENCE TO FB_CoverControl;
	fbBrake				: REFERENCE TO FB_HydraulicsControl;
	fbHydraulics		: REFERENCE TO FB_HydraulicsControl;
	fbFocus		 		: REFERENCE TO FB_FocusControl;
	fbElevation			: REFERENCE TO FB_ElevationControl;
	fbAzimuth	 		: REFERENCE TO FB_AzimuthControl;
	fbDerotator			: REFERENCE TO FB_DerotatorControl;
	fbTelescope			: REFERENCE TO FB_AltAzTelescopeControl;	
END_VAR
VAR
	fbComm				: I_Comm;

	// program selection of the pendant control
	Selection:	UINT;
	// error on the pendant control
	Error:		BOOL;
	horn:			BOOL;
	fbStartTrigger			: R_TRIG;
	DerotatorEnable:	FB_ButtonEnable;
	ElevationEnable: 	FB_ButtonEnable;
	AzimuthEnable: 		FB_ButtonEnable;
	TelescopeControlEnable: 	FB_ButtonEnable;
	TrackingEnable:			FB_ButtonEnable;
	ResetDelay:	TON;
	TwinCATRestart: TC_Restart;
	up_trigger:	R_TRIG;
	down_trigger:	R_TRIG;	
	// manual or automatic operation of the telescope
	telescope_mode : E_TelescopeMode;
	
	reset_trigger		: R_TRIG;

	//DIN17 2.0
	BCD0		AT%I*: BOOL;
	//DIN18 2.1
	BCD2		AT%I*: BOOL;
	//DIN19 2.2
	BCD4		AT%I*: BOOL;
	//DIN20 2.3
	BCD8		AT%I*: BOOL;
	//DIN21 2.4
	reset_switch	AT%I*: BOOL;
	//DIN22 2.5
	direction_up	AT%I*: BOOL;
	//DIN23 2.6
	direction_down	AT%I*: BOOL;
	//DIN24 2.7
	key_switch		AT%I*: BOOL;
	//DIN25 3.0 (enable)
	start_switch	AT%I*: BOOL;
	//DIN26 3.1
	direction_left	AT%I*: BOOL;
	//DIN27 3.2
	direction_right	AT%I*: BOOL;
	
	// Outputs
	
	//DOUT9 1.0
	lamp_up			AT%Q*: BOOL;
	//DOUT10 1.1
	lamp_down			AT%Q*: BOOL;
	//DOUT11 1.2
	lamp_right			AT%Q*: BOOL;
	//DOUT12 1.3
	lamp_left			AT%Q*: BOOL;
	//DOUT13 1.4
	lamp_error			AT%Q*: BOOL;	
	GVL_Telescope: INT;
END_VAR

(* 
This program is responsible for the manual control of the telescope.
all movable parts can be controlled from here. This is mainly for testing and
maintenance.
WARNING! Some of the safety routines are disabled, when operating the telescope manually.
*)
// calculate the value of the selector
Selection := 1*BOOL_TO_UINT(BCD0) + 
			 2*BOOL_TO_UINT(BCD2) + 
			 4*BOOL_TO_UINT(BCD4) +
			 8*BOOL_TO_UINT(BCD8);

// detect disconnection of the manual controls (should also trigger emergency stop).			 
Error := (Selection = 0);

// disable all the lamps
lamp_left := FALSE;
lamp_right := FALSE;
lamp_up := FALSE;
lamp_down := FALSE;
horn := FALSE;

up_trigger(CLK := direction_up);
down_trigger(CLK := direction_down);
//R_Enable(CLK := enable);
// the error lamp is the same as the error lamp of the main panel
lamp_error := lamp_error;


// determine the operation of the telescope based on the switch set
IF key_switch THEN
	telescope_mode := E_TelescopeMode.manual;
ELSE
	telescope_mode := E_TelescopeMode.automatic;
END_IF

// reset or start pushed?
reset_trigger(CLK := reset_switch);
fbStartTrigger(CLK := start_switch);

// enable only the selected item and connect lamps and buttons accordingly
CASE Selection OF
	1, 2, 3:	// reserved for Cover 1-3 control
		lamp_up := fbCovers.IabCoverOpen[Selection];
		lamp_down := fbCovers.IabCoverClosed[Selection];
		IF key_switch THEN
			fbCovers.OabOpenCover[Selection] := direction_up AND fbCovers.IabCoverOpen[Selection];
			fbCovers.OabCloseCover[Selection] := direction_down AND fbCovers.IabCoverClosed[Selection];
			lamp_error := fbCovers.abCoverError[Selection];	
		ELSE
			IF direction_down THEN 
				fbCovers.Close();
			ELSIF direction_up THEN
				fbCovers.Open();
			END_IF		
		END_IF
		
	4:	// Nasmyth / mirror M3 control
		
	5:	// Focus Control
		IF __ISVALIDREF(fbFocus) THEN
			lamp_up := fbFocus.Ready AND NOT fbFocus.InPosLimit;
			lamp_down := fbFocus.Ready AND NOT fbFocus.InNegLimit;
			IF key_switch THEN
				IF fbStartTrigger.Q THEN
					fbFocus.Enable := NOT fbFocus.Enable;
				END_IF
				fbFocus.MovePos := direction_up;
				fbFocus.MoveNeg := direction_down;
				IF reset_trigger.Q THEN
					fbFocus.Reset();
				END_IF
				lamp_error := fbFocus.Error;
			END_IF
		END_IF
							
	6:	// Derotator control
		lamp_left  := fbDerotator.Ready AND NOT fbDerotator.InNegLimit;
		lamp_right := fbDerotator.Ready AND NOT fbDerotator.InPosLimit;
		IF key_switch THEN
			DerotatorEnable(SET := start_switch, Q := fbDerotator.bEnable);
			fbDerotator.MoveNeg := direction_left AND NOT fbDerotator.inDigitalInputs.1;
			fbDerotator.MovePos := direction_right AND NOT fbDerotator.inDigitalInputs.0;
			fbDerotator.bReset := reset_switch;
			lamp_error := fbDerotator.Error;
		END_IF
							
	7:	// Elevation Control
		
		fbElevation.MovePos := direction_up AND fbElevation.inDigitalInputs.0;
		fbElevation.MoveNeg := direction_down AND fbElevation.inDigitalInputs.1;
		IF key_switch THEN
			ElevationEnable(
				SET := start_switch, 
				Q := fbElevation.bEnable);	
		END_IF
		fbElevation.bReset := reset_switch;
		lamp_up := fbElevation.inDigitalInputs.0;
		lamp_down := fbElevation.inDigitalInputs.1;
		lamp_error := fbElevation.bError;
		
	8:	// Azimuth Control
		lamp_left := fbAzimuth.inDigitalInputs.0; // NOT GVL_Telescope.azimut_limit_switch;
		lamp_right := fbAzimuth.inDigitalInputs.1; // NOT GVL_Telescope.azimut_limit_switch;
		fbAzimuth.MoveNeg := direction_left AND fbAzimuth.inDigitalInputs.0;
		fbAzimuth.MovePos := direction_right AND fbAzimuth.inDigitalInputs.1;
		fbAzimuth.bReset := reset_switch;
		IF key_switch THEN
			AzimuthEnable(
				SET := start_switch, 
				Q := fbAzimuth.bEnable);
			lamp_error := fbAzimuth.Error;
		END_IF
		
	9: 	// Dome control
		
	10:	// FilterWheel control
		
	11: lamp_up := fbElevation.fTorque > 0.0;
		lamp_down := fbElevation.fTorque < 0.0;
		
	12:	// manual Telescope Control
		IF key_switch THEN
			lamp_up := fbTelescope.bPower;
			lamp_down := fbTelescope.bPower;
			lamp_left := fbTelescope.bPower;
			lamp_right := fbTelescope.bPower;
	
			fbTelescope.bGoHome := direction_down;
			fbTelescope.bPark := direction_up;
			fbTelescope.bGoto := direction_right;
			TrackingEnable(SET := start_switch, 
							RESET := reset_switch, 
							Q := fbTelescope.bTrack);
			fbTelescope.bReset := reset_switch;
			fbTelescope.bStop := direction_left;	
			lamp_error := fbTelescope.bError;
		END_IF
		
	13: // Telescope Control
		TelescopeControlEnable(
			SET := start_switch, 
			Q := fbTelescope.bPower);
		fbTelescope.bReset := reset_switch;
		IF key_switch THEN
			lamp_up := fbElevation.inDigitalInputs.0;
			lamp_down := fbElevation.inDigitalInputs.1;
			lamp_left := fbAzimuth.inDigitalInputs.0;
			lamp_right := fbAzimuth.inDigitalInputs.1;
			fbElevation.MovePos := direction_up AND fbElevation.inDigitalInputs.0;
			fbElevation.MoveNeg := direction_down AND fbElevation.inDigitalInputs.1;
			fbAzimuth.MoveNeg := direction_left AND fbAzimuth.inDigitalInputs.0;
			fbAzimuth.MovePos := direction_right AND fbAzimuth.inDigitalInputs.1;
			fbTelescope.fRightAscension := fbTelescope.fRightAscensionCalc;
			fbTelescope.fDeclination := fbTelescope.fDeclinationCalc;
		ELSE
			lamp_up := fbElevation.bEnable;
			lamp_down := fbElevation.bEnable;
			lamp_left := fbAzimuth.bEnable;
			lamp_right := fbAzimuth.bEnable;
			IF direction_up THEN 
				fbTelescope.fElevationOffset := fbTelescope.fElevationOffset + 10.0/3600.0; 
			ELSIF direction_down THEN 
				fbTelescope.fElevationOffset := fbTelescope.fElevationOffset - 10.0/3600.0; 
			END_IF;
			IF direction_left THEN 
				fbTelescope.fAzimuthOffset := fbTelescope.fAzimuthOffset - 10.0/3600.0; 
			ELSIF direction_right THEN 
				fbTelescope.fAzimuthOffset := fbTelescope.fAzimuthOffset + 10.0/3600.0; 
			END_IF;
		END_IF
		ResetDelay(IN := reset_switch, PT := T#3S);
		// wait for suction pump to stop
		TwinCATRestart(NETID := '', RESTART := ResetDelay.Q AND NOT fbHydraulics.SuctionRunning, TMOUT := T#60S);
	
	14: horn := key_switch;
		lamp_up := key_switch;
		lamp_down := key_switch;
		lamp_left := key_switch;
		lamp_right := key_switch;
	
	15:	// Hydraulics control
		lamp_up := fbHydraulics.OilPressureOK AND NOT fbBrake.BrakeOpen;
		lamp_down := fbHydraulics.OilPressureOK AND fbBrake.BrakeOpen;
		lamp_left := fbHydraulics.PumpRunning;
		lamp_right := fbHydraulics.SuctionRunning;
		IF key_switch THEN
			IF fbStartTrigger.Q THEN
				fbHydraulics.Enable := NOT fbHydraulics.Enable;
			END_IF
			IF reset_trigger.Q THEN
				fbHydraulics.Reset();
			END_IF
			
			IF direction_up THEN
				fbBrake.OpenBrake();
			END_IF
			IF direction_down THEN
				fbBrake.CloseBrake();
			END_IF
			fbHydraulics.ManualStartSuction := direction_right;
			fbHydraulics.ManualStopPump := direction_left;
			lamp_error := fbHydraulics.Error;
		END_IF
END_CASE

//FB_Init is always available implicitly and it is used primarily for initialization.
//The return value is not evaluated. For a specific influence, you can also declare the
//methods explicitly and provide additional code there with the standard initialization
//code. You can evaluate the return value.
METHOD FB_Init: BOOL
VAR_INPUT
    bInitRetains: BOOL; // TRUE: the retain variables are initialized (reset warm / reset cold)
    bInCopyCode: BOOL;  // TRUE: the instance will be copied to the copy code afterward (online change)
	comm			: I_Comm;   
END_VAR
THIS^.fbComm 	:= comm;
END_METHOD

END_FUNCTION_BLOCK

// ---- POUs/FB_TelescopeAuxiliary.TcPOU
FUNCTION_BLOCK FB_TelescopeAuxiliary
VAR
	MQTTTimer : TON := (PT:=T#5S);
	tempSensorM2		AT%I*: INT;	// BT9 mirror
	tempSensorM1		AT%I*: INT;	// // BT10
END_VAR
VAR_INPUT
	comm: I_Comm;
END_VAR
VAR_OUTPUT
	// BT9 mirror
	temperature_mirror2:	REAL;
	// BT10
	temperature_mirror1:	REAL;
END_VAR

//temperature_mirror1 := GVL_Telescope.temperature_mirror1 / 1000.0;
//temperature_mirror2 := GVL_Telescope.temperature_mirror2 / 1000.0;
temperature_mirror1 := tempSensorM1 / 32767.0 * 150.0 - 50.0;
temperature_mirror2 := tempSensorM2 / 32767.0 * 150.0 - 50.0;

MQTTTimer(IN:=TRUE);
IF MQTTTimer.Q THEN // publish new payload every second

	comm.Publish('telescope', 'dome', 'Mirror1Temperature',	LREAL_TO_FMTSTR(temperature_mirror1, 2, TRUE));
	comm.Publish('telescope', 'dome', 'Mirror2Temperature',	LREAL_TO_FMTSTR(temperature_mirror2, 2, TRUE));
	
	MQTTTimer(IN:=FALSE);

END_IF

END_FUNCTION_BLOCK

// ---- GlobalTextList.TcGTLO
TEXTLIST GlobalTextList
  541 = '%.0f'
  332 = '%.0f%'
  390 = '%.1f %'
  580 = '%.1f mm'
  730 = '%.2f mm'
  1120 = '%.2f °'
  943 = '%.2f °/s'
  144 = '%.4f '
  339 = '%.4f mm'
  848 = '%.4f °'
  78 = '+'
  114 = '-'
  248 = 'Axis +'
  375 = 'Axis -'
  785 = 'Azimuth:'
  247 = 'Brake'
  911 = 'Brake clearing'
  798 = 'Brake closed'
  396 = 'Brake open'
  958 = 'Brakes'
  121 = 'Brakes closed'
  883 = 'Brakes open'
  688 = 'Calibrated'
  772 = 'Close'
  41 = 'Close brake'
  499 = 'Close brakes'
  10 = 'Closed'
  392 = 'Cold'
  12 = 'Cover 1'
  822 = 'Cover 1\\'
  678 = 'Cover 2'
  857 = 'Cover 3'
  816 = 'Current'
  815 = 'Derotator:'
  524 = 'Diag: %s'
  101 = 'EL1904'
  761 = 'EL2904'
  409 = 'Elevation:'
  894 = 'Enable'
  377 = 'ErrAck'
  421 = 'Error'
  225 = 'Estop: %s'
  755 = 'Far'
  488 = 'Global'
  331 = 'High'
  483 = 'Homing'
  81 = 'Hot'
  163 = 'Level'
  846 = 'Level:'
  557 = 'Limits'
  58 = 'Low'
  697 = 'Manual'
  564 = 'Move'
  99 = 'Moving'
  59 = 'Near'
  648 = 'Offset +'
  779 = 'Offset -'
  33 = 'Oil cold'
  995 = 'Oil high'
  856 = 'Oil hot'
  768 = 'Oil low'
  37 = 'Oil pan maximum'
  481 = 'Oil pressure OK'
  874 = 'Oil Status'
  498 = 'Oil warning'
  727 = 'Open'
  482 = 'Open brake'
  868 = 'Open brakes'
  744 = 'Override Start Sucction'
  606 = 'Override stop pump'
  890 = 'Overrides'
  384 = 'Pan max'
  645 = 'Pan maximum'
  295 = 'Position'
  641 = 'Pressure'
  540 = 'Pressure OK'
  196 = 'Pump'
  523 = 'Pump running'
  176 = 'Ready'
  695 = 'Reset'
  789 = 'Restart'
  521 = 'Safety Diag: %s'
  672 = 'Safety State: %s'
  309 = 'Set'
  566 = 'Start'
  202 = 'Start Sucction'
  27 = 'Start suction'
  809 = 'State: %s'
  677 = 'Status'
  328 = 'STO ErrAck:'
  376 = 'STO:'
  189 = 'Stop pump'
  614 = 'Sucction'
  782 = 'Sucction running'
  552 = 'Suction'
  136 = 'Unlocked'
  67 = 'Velocity'
  194 = 'Warning'
END_TEXTLIST

// ---- VISUs/Azimuth.TcVIS
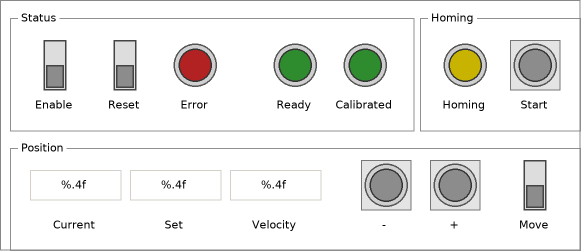
VISUALIZATION Azimuth  // 581x251
    GroupBox (10,10 404x121), "Status"
        DipSwitch (20,30 50x50), variable: MAIN.AzimuthControl.bEnable, behaviour: TOGGLE, style: Switch-DipSwitch-Gray
        DipSwitch (90,30 50x50), variable: MAIN.AzimuthControl.bReset, behaviour: TOGGLE, style: Switch-DipSwitch-Gray
        Lamp1 (160,30 50x50), variable: MAIN.AzimuthControl.bError, style: Lamp-Lamp1-Red
        Lamp1 (260,30 50x50), variable: MAIN.AzimuthControl.bReady, style: Lamp-Lamp1-Green
        Lamp1 (330,30 50x50), variable: MAIN.AzimuthControl.bCalibrated, style: Lamp-Lamp1-Green
        Label (10,80 68x30), "Enable"
        Label (80,80 68x30), "Reset"
        Label (150,80 68x30), "Error"
        Label (250,80 68x30), "Ready"
        Label (320,80 68x30), "Calibrated"
    GroupBox (420,10 161x121), "Homing"
        Lamp1 (20,30 50x50), variable: MAIN.AzimuthControl.bHomeAxis, style: Lamp-Lamp1-Yellow
        Label (10,80 68x30), "Homing"
        PushSwitch (90,30 50x50), variable: MAIN.AzimuthControl.bHomeAxis, behaviour: TOGGLE, style: Switch-PushSwitch-Gray
        Label (80,80 68x30), "Start"
    GroupBox (10,140 571x111), "Position"
        Textfield (20,30 91x30), "%.4f", text variable: MAIN.AzimuthControl.fActualPosition
        Label (30,70 68x30), "Current"
        Textfield (120,30 91x30), "%.4f", text variable: MAIN.AzimuthControl.fPosition
            OnMouseUp: write the text variable via InputWithLimits, min MAIN.AzimuthControl.fMinPosition, max MAIN.AzimuthControl.fMaxPosition
        Textfield (220,30 91x30), "%.4f", text variable: MAIN.AzimuthControl.fVelocity
            OnMouseUp: write the text variable via InputWithLimits, min 0, max 200
        PushSwitch (351,20 50x50), variable: MAIN.AzimuthControl.bMoveNeg, behaviour: TOGGLE, style: Switch-PushSwitch-Gray
        PushSwitch (420,20 50x50), variable: MAIN.AzimuthControl.bMovePos, behaviour: TOGGLE, style: Switch-PushSwitch-Gray
        DipSwitch (500,20 50x50), variable: MAIN.AzimuthControl.bMoveAxis, behaviour: TOGGLE, style: Switch-DipSwitch-Gray
        Label (340,70 68x30), "-"
        Label (410,70 68x30), "+"
        Label (490,70 68x30), "Move"
    Label (140,210 68x30), "Set"
    Label (240,210 68x30), "Velocity"
END_VISUALIZATION

// ---- VISUs/Cover.TcVIS
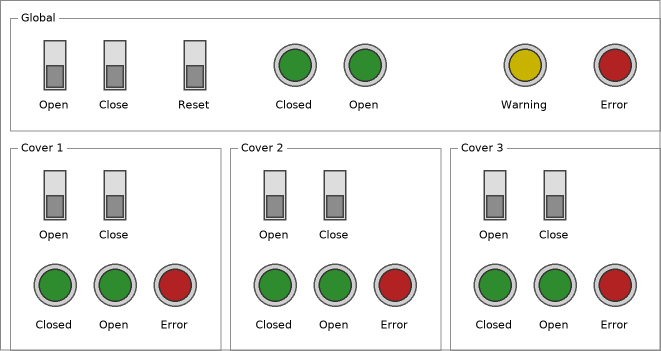
VISUALIZATION Cover  // 661x351
    GroupBox (10,10 651x121), "Global"
        DipSwitch (20,30 50x50), variable: MAIN.AzimuthControl.bEnable, behaviour: TOGGLE, style: Switch-DipSwitch-Gray
        DipSwitch (80,30 50x50), variable: MAIN.AzimuthControl.bReset, behaviour: TOGGLE, style: Switch-DipSwitch-Gray
        Lamp1 (260,30 50x50), variable: MAIN.AzimuthControl.bReady, style: Lamp-Lamp1-Green
        Lamp1 (330,30 50x50), variable: MAIN.AzimuthControl.bCalibrated, style: Lamp-Lamp1-Green
        Label (10,80 68x30), "Open"
        Label (70,80 68x30), "Close"
        Label (250,80 68x30), "Closed"
        Label (320,80 68x30), "Open"
        DipSwitch (160,30 50x50), variable: MAIN.AzimuthControl.bReset, behaviour: TOGGLE, style: Switch-DipSwitch-Gray
        Lamp1 (490,30 50x50), variable: MAIN.AzimuthControl.bHomeAxis, style: Lamp-Lamp1-Yellow
        Lamp1 (580,30 50x50), style: Lamp-Lamp1-Red
        Label (570,80 68x30), "Error"
        Label (480,80 68x30), "Warning"
    GroupBox (10,140 211x211), "Cover 1"
        Label (130,170 68x30), "Error"
        Lamp1 (20,120 50x50), variable: MAIN.CoverControl.abCoverClosed[1], style: Lamp-Lamp1-Green
        Lamp1 (80,120 50x50), variable: MAIN.CoverControl.abCoverOpen[1], style: Lamp-Lamp1-Green
        Label (10,170 68x30), "Closed"
        Label (70,170 68x30), "Open"
        DipSwitch (20,30 50x50), variable: MAIN.CoverControl.OabOpenCover[1], behaviour: TOGGLE, style: Switch-DipSwitch-Gray
        DipSwitch (80,30 50x50), variable: MAIN.CoverControl.OabCloseCover[1], behaviour: TOGGLE, style: Switch-DipSwitch-Gray
        Label (10,80 68x30), "Open"
        Label (70,80 68x30), "Close"
        Lamp1 (140,120 50x50), variable: MAIN.CoverControl.abCoverError[1], style: Lamp-Lamp1-Red
    Label (160,90 68x30), "Reset"
    GroupBox (230,140 211x211), "Cover 2"
        Label (130,170 68x30), "Error"
        Lamp1 (20,120 50x50), variable: MAIN.CoverControl.abCoverClosed[2], style: Lamp-Lamp1-Green
        Lamp1 (80,120 50x50), variable: MAIN.CoverControl.abCoverOpen[2], style: Lamp-Lamp1-Green
        Label (10,170 68x30), "Closed"
        Label (70,170 68x30), "Open"
        DipSwitch (20,30 50x50), variable: MAIN.CoverControl.OabOpenCover[2], behaviour: TOGGLE, style: Switch-DipSwitch-Gray
        DipSwitch (80,30 50x50), variable: MAIN.CoverControl.OabCloseCover[2], behaviour: TOGGLE, style: Switch-DipSwitch-Gray
        Label (10,80 68x30), "Open"
        Label (70,80 68x30), "Close"
        Lamp1 (140,120 50x50), variable: MAIN.CoverControl.abCoverError[2], style: Lamp-Lamp1-Red
    GroupBox (450,140 211x211), "Cover 3"
        Label (130,170 68x30), "Error"
        Lamp1 (20,120 50x50), variable: MAIN.CoverControl.abCoverClosed[3], style: Lamp-Lamp1-Green
        Lamp1 (80,120 50x50), variable: MAIN.CoverControl.abCoverOpen[3], style: Lamp-Lamp1-Green
        Label (10,170 68x30), "Closed"
        Label (70,170 68x30), "Open"
        DipSwitch (20,30 50x50), variable: MAIN.CoverControl.OabOpenCover[3], behaviour: TOGGLE, style: Switch-DipSwitch-Gray
        DipSwitch (80,30 50x50), variable: MAIN.CoverControl.OabCloseCover[3], behaviour: TOGGLE, style: Switch-DipSwitch-Gray
        Label (10,80 68x30), "Open"
        Label (70,80 68x30), "Close"
        Lamp1 (140,120 50x50), variable: MAIN.CoverControl.abCoverError[3], style: Lamp-Lamp1-Red
END_VISUALIZATION

// ---- VISUs/Derotator.TcVIS
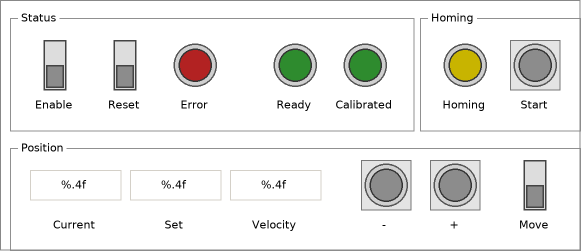
VISUALIZATION Derotator  // 581x251
    GroupBox (10,10 404x121), "Status"
        DipSwitch (20,30 50x50), variable: MAIN.DerotatorControl.bEnable, behaviour: TOGGLE, style: Switch-DipSwitch-Gray
        DipSwitch (90,30 50x50), variable: MAIN.DerotatorControl.bReset, behaviour: TOGGLE, style: Switch-DipSwitch-Gray
        Lamp1 (160,30 50x50), variable: MAIN.DerotatorControl.bError, style: Lamp-Lamp1-Red
        Lamp1 (260,30 50x50), variable: MAIN.DerotatorControl.bReady, style: Lamp-Lamp1-Green
        Lamp1 (330,30 50x50), variable: MAIN.DerotatorControl.bCalibrated, style: Lamp-Lamp1-Green
        Label (10,80 68x30), "Enable"
        Label (80,80 68x30), "Reset"
        Label (150,80 68x30), "Error"
        Label (250,80 68x30), "Ready"
        Label (320,80 68x30), "Calibrated"
    GroupBox (420,10 161x121), "Homing"
        Lamp1 (20,30 50x50), variable: MAIN.DerotatorControl.bHomeAxis, style: Lamp-Lamp1-Yellow
        Label (10,80 68x30), "Homing"
        PushSwitch (90,30 50x50), variable: MAIN.DerotatorControl.bHomeAxis, behaviour: TOGGLE, style: Switch-PushSwitch-Gray
        Label (80,80 68x30), "Start"
    GroupBox (10,140 571x111), "Position"
        Textfield (20,30 91x30), "%.4f", text variable: MAIN.DerotatorControl.fActualPosition
        Label (30,70 68x30), "Current"
        Textfield (120,30 91x30), "%.4f", text variable: MAIN.DerotatorControl.fPosition
            OnMouseUp: write the text variable via InputWithLimits, min MAIN.DerotatorControl.fMinPosition, max MAIN.DerotatorControl.fMaxPosition
        Textfield (220,30 91x30), "%.4f", text variable: MAIN.DerotatorControl.fVelocity
            OnMouseUp: write the text variable via InputWithLimits, min 0, max 200
        PushSwitch (351,20 50x50), variable: MAIN.DerotatorControl.bMoveNeg, behaviour: TOGGLE, style: Switch-PushSwitch-Gray
        PushSwitch (420,20 50x50), variable: MAIN.DerotatorControl.bMovePos, behaviour: TOGGLE, style: Switch-PushSwitch-Gray
        DipSwitch (500,20 50x50), variable: MAIN.DerotatorControl.bMoveAxis, behaviour: TOGGLE, style: Switch-DipSwitch-Gray
        Label (340,70 68x30), "-"
        Label (410,70 68x30), "+"
        Label (490,70 68x30), "Move"
    Label (140,210 68x30), "Set"
    Label (240,210 68x30), "Velocity"
END_VISUALIZATION

// ---- VISUs/Elevation.TcVIS
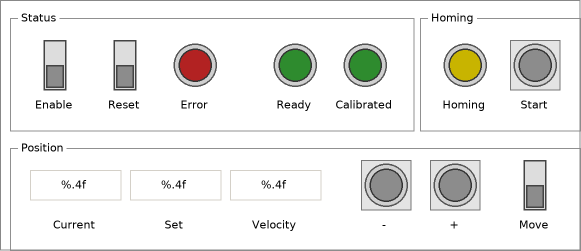
VISUALIZATION Elevation  // 581x251
    GroupBox (10,10 404x121), "Status"
        DipSwitch (20,30 50x50), variable: MAIN.ElevationControl.bEnable, behaviour: TOGGLE, style: Switch-DipSwitch-Gray
        DipSwitch (90,30 50x50), variable: MAIN.ElevationControl.bReset, behaviour: TOGGLE, style: Switch-DipSwitch-Gray
        Lamp1 (160,30 50x50), variable: MAIN.ElevationControl.bError, style: Lamp-Lamp1-Red
        Lamp1 (260,30 50x50), variable: MAIN.ElevationControl.bReady, style: Lamp-Lamp1-Green
        Lamp1 (330,30 50x50), variable: MAIN.ElevationControl.bCalibrated, style: Lamp-Lamp1-Green
        Label (10,80 68x30), "Enable"
        Label (80,80 68x30), "Reset"
        Label (150,80 68x30), "Error"
        Label (250,80 68x30), "Ready"
        Label (320,80 68x30), "Calibrated"
    GroupBox (420,10 161x121), "Homing"
        Lamp1 (20,30 50x50), variable: MAIN.ElevationControl.bHomeAxis, style: Lamp-Lamp1-Yellow
        Label (10,80 68x30), "Homing"
        PushSwitch (90,30 50x50), variable: MAIN.ElevationControl.bHomeAxis, behaviour: TOGGLE, style: Switch-PushSwitch-Gray
        Label (80,80 68x30), "Start"
    GroupBox (10,140 571x111), "Position"
        Textfield (20,30 91x30), "%.4f", text variable: MAIN.ElevationControl.fActualPosition
        Label (30,70 68x30), "Current"
        Textfield (120,30 91x30), "%.4f", text variable: MAIN.ElevationControl.fPosition
            OnMouseUp: write the text variable via InputWithLimits, min MAIN.ElevationControl.fMinPosition, max MAIN.ElevationControl.fMaxPosition
        Textfield (220,30 91x30), "%.4f", text variable: MAIN.ElevationControl.fVelocity
            OnMouseUp: write the text variable via InputWithLimits, min 0, max 200
        PushSwitch (351,20 50x50), variable: MAIN.ElevationControl.bMoveNeg, behaviour: TOGGLE, style: Switch-PushSwitch-Gray
        PushSwitch (420,20 50x50), variable: MAIN.ElevationControl.bMovePos, behaviour: TOGGLE, style: Switch-PushSwitch-Gray
        DipSwitch (500,20 50x50), variable: MAIN.ElevationControl.bMoveAxis, behaviour: TOGGLE, style: Switch-DipSwitch-Gray
        Label (340,70 68x30), "-"
        Label (410,70 68x30), "+"
        Label (490,70 68x30), "Move"
    Label (140,210 68x30), "Set"
    Label (240,210 68x30), "Velocity"
END_VISUALIZATION

// ---- VISUs/Focus.TcVIS
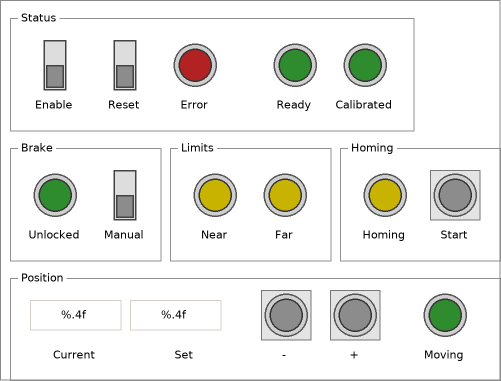
VISUALIZATION Focus  // 501x381
    GroupBox (10,10 404x121), "Status"
        DipSwitch (20,30 50x50), variable: MAIN.FocusControl.bEnable, behaviour: TOGGLE, style: Switch-DipSwitch-Gray
        DipSwitch (90,30 50x50), variable: MAIN.FocusControl.bReset, behaviour: TOGGLE, style: Switch-DipSwitch-Gray
        Lamp1 (160,30 50x50), variable: MAIN.FocusControl.bError, style: Lamp-Lamp1-Red
        Lamp1 (260,30 50x50), variable: MAIN.FocusControl.bReady, style: Lamp-Lamp1-Green
        Lamp1 (330,30 50x50), variable: MAIN.FocusControl.bCalibrated, style: Lamp-Lamp1-Green
        Label (10,80 68x30), "Enable"
        Label (80,80 68x30), "Reset"
        Label (150,80 68x30), "Error"
        Label (250,80 68x30), "Ready"
        Label (320,80 68x30), "Calibrated"
        Lamp1 (410,280 50x50), variable: MAIN.AzimuthControl.bCalibrated, style: Lamp-Lamp1-Green
    GroupBox (340,140 161x121), "Homing"
        Lamp1 (20,30 50x50), variable: MAIN.FocusControl.bHomeAxis, style: Lamp-Lamp1-Yellow
        Label (10,80 68x30), "Homing"
        PushSwitch (90,30 50x50), variable: MAIN.FocusControl.bHomeAxis, behaviour: TOGGLE, style: Switch-PushSwitch-Gray
        Label (80,80 68x30), "Start"
    GroupBox (10,140 151x121), "Brake"
        DipSwitch (90,30 50x50), variable: MAIN.FocusControl.bManualUnlock, behaviour: TOGGLE, style: Switch-DipSwitch-Gray
        Lamp1 (20,30 50x50), variable: MAIN.FocusControl.bFocusUnlocked, style: Lamp-Lamp1-Green
        Label (80,80 68x30), "Manual"
        Label (10,80 68x30), "Unlocked"
    GroupBox (170,140 161x121), "Limits"
        Lamp1 (20,30 50x50), variable: MAIN.FocusControl.InNegLimit, style: Lamp-Lamp1-Yellow
        Label (10,80 68x30), "Near"
        Lamp1 (90,30 50x50), variable: MAIN.FocusControl.InPosLimit, style: Lamp-Lamp1-Yellow
    Label (250,220 68x30), "Far"
    GroupBox (10,270 491x111), "Position"
        Textfield (20,30 91x30), "%.4f", text variable: MAIN.FocusControl.fActualPosition
        Label (30,70 68x30), "Current"
        Textfield (120,30 91x30), "%.4f", text variable: MAIN.FocusControl.fPosition
            OnMouseUp: write the text variable via InputWithLimits, min MAIN.AzimuthControl.fMinPosition, max MAIN.AzimuthControl.fMaxPosition
        PushSwitch (251,20 50x50), variable: MAIN.FocusControl.bMoveNeg, behaviour: TOGGLE, style: Switch-PushSwitch-Gray
        PushSwitch (320,20 50x50), variable: MAIN.FocusControl.MovePos, behaviour: TOGGLE, style: Switch-PushSwitch-Gray
        Label (240,70 68x30), "-"
        Label (310,70 68x30), "+"
        Label (140,70 68x30), "Set"
        Lamp1 (410,20 50x50), variable: MAIN.FocusControl.bMoveAxis, style: Lamp-Lamp1-Green
    Label (410,340 68x30), "Moving"
END_VISUALIZATION

// ---- VISUs/Hydraulics.TcVIS
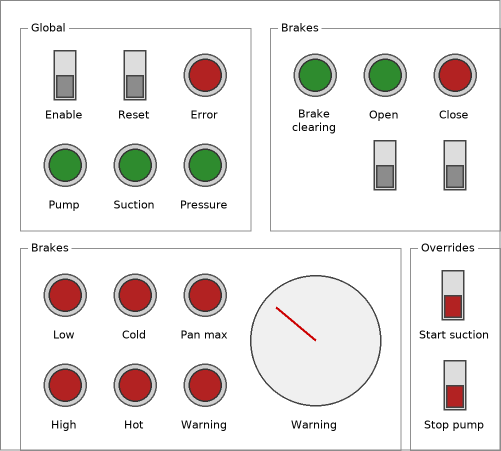
VISUALIZATION Hydraulics  // 501x451
4096VAR_IN_OUT
	
END_VAR
    GroupBox (20,20 231x211), "Global"
        DipSwitch (20,30 50x50), variable: MAIN.HydraulicsControl.bEnable, behaviour: TOGGLE, style: Switch-DipSwitch-Gray
        DipSwitch (90,30 50x50), variable: MAIN.HydraulicsControl.bReset, behaviour: TOGGLE, style: Switch-DipSwitch-Gray
        Lamp1 (160,30 50x50), variable: MAIN.HydraulicsControl.bError, style: Lamp-Lamp1-Red
        Lamp1 (20,120 50x50), variable: MAIN.HydraulicsControl.bPumpRunning, style: Lamp-Lamp1-Green
        Lamp1 (90,120 50x50), variable: MAIN.HydraulicsControl.bSuctionRunning, style: Lamp-Lamp1-Green
        Label (10,80 68x30), "Enable"
        Label (80,80 68x30), "Reset"
        Label (150,80 68x30), "Error"
        Label (10,170 68x30), "Pump"
        Label (80,170 68x30), "Suction"
        Lamp1 (160,120 50x50), variable: MAIN.HydraulicsControl.bOilPressureOK, style: Lamp-Lamp1-Green
        Label (150,170 68x30), "Pressure"
    GroupBox (270,20 231x211), "Brakes"
        DipSwitch (90,120 50x50), variable: MAIN.HydraulicsControl.bOpenBrake, behaviour: TOGGLE, style: Switch-DipSwitch-Gray
        DipSwitch (160,120 50x50), variable: MAIN.HydraulicsControl.bCloseBrake, behaviour: TOGGLE, style: Switch-DipSwitch-Gray
        Lamp1 (160,30 50x50), variable: MAIN.HydraulicsControl.bBrakeClosed, style: Lamp-Lamp1-Red
        Lamp1 (20,30 50x50), variable: MAIN.HydraulicsControl.bBrakeClearing, style: Lamp-Lamp1-Green
        Label (150,80 68x30), "Close"
        Label (10,80 68x41), "Brake clearing"
        Lamp1 (90,30 50x50), variable: MAIN.HydraulicsControl.bBrakeOpen, style: Lamp-Lamp1-Green
        Label (80,80 68x30), "Open"
    GroupBox (20,240 381x211), "Brakes"
        Lamp1 (160,30 50x50), variable: MAIN.HydraulicsControl.bOilPanMaximum, style: Lamp-Lamp1-Red
        Label (150,80 68x30), "Pan max"
        Lamp1 (20,30 50x50), variable: MAIN.HydraulicsControl.bOilLow, style: Lamp-Lamp1-Red
        Lamp1 (90,30 50x50), variable: MAIN.HydraulicsControl.bOilCold, style: Lamp-Lamp1-Red
        Label (80,80 68x30), "Cold"
        Label (10,80 68x30), "Low"
        Lamp1 (160,120 50x50), variable: MAIN.HydraulicsControl.bOilWarning, style: Lamp-Lamp1-Red
        Meter360 (230,30 131x141), value: MAIN.HydraulicsControl.fOilLevel, style: Meter-Meter360-Gray, scale format: %.0f, scale 0..120
        Label (260,170 68x30), "Warning"
    Label (170,410 68x30), "Warning"
    Lamp1 (40,360 50x50), variable: MAIN.HydraulicsControl.bOilHigh, style: Lamp-Lamp1-Red
    Lamp1 (110,360 50x50), variable: MAIN.HydraulicsControl.bOilHot, style: Lamp-Lamp1-Red
    Label (100,410 68x30), "Hot"
    Label (30,410 68x30), "High"
    GroupBox (410,240 91x211), "Overrides"
        DipSwitch (18,30 50x50), variable: MAIN.HydraulicsControl.bManualSuction, behaviour: TOGGLE, style: Switch-DipSwitch-Red
        DipSwitch (20,120 50x50), variable: MAIN.HydraulicsControl.bManualPumpStop, behaviour: TOGGLE, style: Switch-DipSwitch-Red
        Label (10,80 68x30), "Start suction"
        Label (10,170 68x30), "Stop pump"
END_VISUALIZATION
